CONFIGURATION Untitled1
  RESOURCE Untitled1 ON PLC
    VAR_GLOBAL  (* INPUTS *)
      ivar_s_Dstartbutton AT %I* : BOOL;
      ivar_s_Dstopbutton AT %I* : BOOL;
      ivar_s_Dresetbutton AT %I* : BOOL;
      ivar_s_Dautoswitch AT %I* : BOOL;
      ivar_s_Din4 AT %I* : BOOL;
      ivar_s_Din5 AT %I* : BOOL;
      ivar_s_Din6 AT %I* : BOOL;
      ivar_s_Din7 AT %I* : BOOL;
      ivar_s_pusher1_in AT %I* : BOOL;
      ivar_s_pusher1_out AT %I* : BOOL;
      ivar_s_stack1filled AT %I* : BOOL;
      ivar_s_product1 AT %I* : BOOL;
      ivar_s_pusher2_in AT %I* : BOOL;
      ivar_s_pusher2_out AT %I* : BOOL;
      ivar_s_stack2filled AT %I* : BOOL;
      ivar_s_product2 AT %I* : BOOL;
      ivar_s_pusher3_in AT %I* : BOOL;
      ivar_s_pusher3_out AT %I* : BOOL;
      ivar_s_stack3filled AT %I* : BOOL;
      ivar_s_product3 AT %I* : BOOL;
      ivar_s_handlingbusy AT %I* : BOOL;
      ivar_s_Hstartbutton AT %I* : BOOL;
      ivar_s_Hstopbutton AT %I* : BOOL;
      ivar_s_Hresetbutton AT %I* : BOOL;
      ivar_s_Hautoswitch AT %I* : BOOL;
      ivar_s_Hin4 AT %I* : BOOL;
      ivar_s_Hin5 AT %I* : BOOL;
      ivar_s_Hin6 AT %I* : BOOL;
      ivar_s_Hin7 AT %I* : BOOL;
      ivar_s_xpos_at1 AT %I* : BOOL;
      ivar_s_xpos_at2 AT %I* : BOOL;
      ivar_s_xpos_at3 AT %I* : BOOL;
      ivar_s_xpos_atdrop AT %I* : BOOL;
      ivar_s_zpos_atup AT %I* : BOOL;
      ivar_s_zpos_atdown AT %I* : BOOL;
      ivar_s_gripper AT %I* : BOOL;
      ivar_s_transfer_atpickup AT %I* : BOOL;
      ivar_s_transfer_atdrop AT %I* : BOOL;
      ivar_s_transfer_athalfway AT %I* : BOOL;
      ivar_s_vacuum AT %I* : BOOL;
      ivar_s_product4 AT %I* : BOOL;
      ivar_s_testingbusy AT %I* : BOOL;
      ivar_s_Tstartbutton AT %I* : BOOL;
      ivar_s_Tstopbutton AT %I* : BOOL;
      ivar_s_Tautoswitch AT %I* : BOOL;
      ivar_s_Tresetbutton AT %I* : BOOL;
      ivar_s_Tin4 AT %I* : BOOL;
      ivar_s_Tin5 AT %I* : BOOL;
      ivar_s_Tin6 AT %I* : BOOL;
      ivar_s_Tin7 AT %I* : BOOL;
      ivar_s_elevator_up AT %I* : BOOL;
      ivar_s_elevator_down AT %I* : BOOL;
      ivar_s_pusher AT %I* : BOOL;
      ivar_s_opticalT AT %I* : BOOL;
      ivar_s_capacitive AT %I* : BOOL;
      ivar_s_reflective AT %I* : BOOL;
      ivar_s_productheight AT %I* : BOOL;
      ivar_s_bufferingbusy AT %I* : BOOL;
      ivar_s_Bstartbutton AT %I* : BOOL;
      ivar_s_Bstopbutton AT %I* : BOOL;
      ivar_s_Bautoswitch AT %I* : BOOL;
      ivar_s_Bresetbutton AT %I* : BOOL;
      ivar_s_Bin4 AT %I* : BOOL;
      ivar_s_Bin5 AT %I* : BOOL;
      ivar_s_Bin6 AT %I* : BOOL;
      ivar_s_Bin7 AT %I* : BOOL;
      ivar_s_atin AT %I* : BOOL;
      ivar_s_atseparator AT %I* : BOOL;
      ivar_s_atend AT %I* : BOOL;
      ivar_s_separator_opened AT %I* : BOOL;
      ivar_s_separator_closed AT %I* : BOOL;
      ivar_s_processingbusy AT %I* : BOOL;
      ivar_s_Pstartbutton AT %I* : BOOL;
      ivar_s_Pstopbutton AT %I* : BOOL;
      ivar_s_Pautoswitch AT %I* : BOOL;
      ivar_s_Presetbutton AT %I* : BOOL;
      ivar_s_Pin4 AT %I* : BOOL;
      ivar_s_Pin5 AT %I* : BOOL;
      ivar_s_Pin6 AT %I* : BOOL;
      ivar_s_Pin7 AT %I* : BOOL;
      ivar_s_atinput AT %I* : BOOL;
      ivar_s_attest AT %I* : BOOL;
      ivar_s_atdrill AT %I* : BOOL;
      ivar_s_atexit AT %I* : BOOL;
      ivar_s_atspare AT %I* : BOOL;
      ivar_s_clamp AT %I* : BOOL;
      ivar_s_test_ok AT %I* : BOOL;
      ivar_s_drill_up AT %I* : BOOL;
      ivar_s_drill_down AT %I* : BOOL;
      ivar_s_turntable AT %I* : BOOL;
      ivar_s_sortingbusy AT %I* : BOOL;
      ivar_s_Sstartbutton AT %I* : BOOL;
      ivar_s_Sstopbutton AT %I* : BOOL;
      ivar_s_Sautoswitch AT %I* : BOOL;
      ivar_s_Sresetbutton AT %I* : BOOL;
      ivar_s_Sin4 AT %I* : BOOL;
      ivar_s_Sin5 AT %I* : BOOL;
      ivar_s_Sin6 AT %I* : BOOL;
      ivar_s_Sin7 AT %I* : BOOL;
      ivar_s_product AT %I* : BOOL;
      ivar_s_inductive AT %I* : BOOL;
      ivar_s_optical AT %I* : BOOL;
      ivar_s_slidefull AT %I* : BOOL;
      ivar_s_gate1_opened AT %I* : BOOL;
      ivar_s_gate1_closed AT %I* : BOOL;
      ivar_s_gate2_opened AT %I* : BOOL;
      ivar_s_gate2_closed AT %I* : BOOL;
    END_VAR
    VAR_GLOBAL  (* TIMERS *)
      timer0 : TON;
      timer1 : TON;
      curTimer : INT := 0;
    END_VAR
    TASK PlcTask(INTERVAL := t#10ms, PRIORITY := 20);
    PROGRAM MAIN WITH PlcTask : MAIN;
  END_RESOURCE
END_CONFIGURATION
